(* CoDeSys 2.3.9.41 project: pogonazh_134_03_R.pro *)
(* Libraries: Util.lib 15.6.21 11:37:35, ПЛК_ПЧВ_v2.lib 17.6.21 09:07:23, STANDARD.LIB 15.6.21 11:37:35, IECSFC.LIB 15.6.21 11:37:35, ANALYZATION.LIB 15.6.21 11:37:35 *)

(* PLC configuration (modules and I/O channels)
InputByte AT %IB0.0 [ByteInput] 8 discrete inputs
DO_1_0 AT %QX1.0 [BitOutput] First
DO_1_1 AT %QX1.1 [BitOutput] Second
DO_2_0 AT %QX2.0 [BitOutput] First
AT %QX2.1 [BitOutput] Second
DO_3_0 AT %QX3.0 [BitOutput] First
DO_3_1 AT %QX3.1 [BitOutput] Second
DO_4_0 AT %QX4.0 [BitOutput] First
DO_4_1 AT %QX4.1 [BitOutput] Second
DO_5_0 AT %QX5.0 [BitOutput] First
DO_5_1 AT %QX5.1 [BitOutput] Second
DO_6_0 AT %QX6.0 [BitOutput] First
DO_6_1 AT %QX6.1 [BitOutput] Second
AT %QX7.0 [BitOutput] Special output
modbusLastAddr AT %QD8.0 [DWordOutput] Last address
modbusLastErr AT %QW8.1 [WordOutput] Last error
RS-485-1 [COM1_USART] node 0, in %IB8.0 out %QB8.0 {CommunicationSpeed = 19200; Parity = NO PARITY CHECK; BitLength = 8 bits; StopLength = One stop bit; InterfaceType = RS485; FrameOriented = RTU; Timeout = 0; Visibility = No}
Universal Modbus device [ID2000] node 1, in %IB8.1 out %QB8.1 {ModuleIP = 10:0:0:223; ServiceTimeout = 150; TCPport = 502; NetMode = Serial; ModuleSlaveAddress = 2; RequestType = By poll time; PeriodOfService = 1000; Visibility = No; RepeatCounter = 2; ByteSequence = Native}
  AT %QB8.1.0 [ComChannel] Command (0xff - Start)
Dist_on_pistol_1 AT %IW8.1.0.0 [WordInput]
Dist_on_pistol_2 AT %IW8.1.1.0 [WordInput]
Dist_on_pistol_3 AT %IW8.1.2.0 [WordInput]
Dist_on_pistol_4 AT %IW8.1.3.0 [WordInput]
Dist_on_pistol_5 AT %IW8.1.4.0 [WordInput]
Dist_on_pistol_6 AT %IW8.1.5.0 [WordInput]
Dist_off_pistol_1 AT %IW8.1.6.0 [WordInput]
Dist_off_pistol_2 AT %IW8.1.7.0 [WordInput]
Dist_off_pistol_3 AT %IW8.1.8.0 [WordInput]
Dist_off_pistol_4 AT %IW8.1.9.0 [WordInput]
Dist_off_pistol_5 AT %IW8.1.10.0 [WordInput]
Dist_off_pistol_6 AT %IW8.1.11.0 [WordInput]
DistOnPistMinimum AT %IW8.1.12.0 [WordInput]
qInvStatusW AT %QW8.1.13.0 [WordOutput]
AT %QB8.2.0 [ComChannel] Command (0xff - Start)
iTP1 AT %IW8.2.0.0 [WordInput]
iTP2 AT %IW8.2.1.0 [WordInput]
iTP3 AT %IW8.2.2.0 [WordInput]
iTP4 AT %IW8.2.3.0 [WordInput]
iTP5 AT %IW8.2.4.0 [WordInput]
iTP6 AT %IW8.2.5.0 [WordInput]
iTPGlob AT %ID8.2.6.0 [FloatInput]
iDate AT %ID8.2.7.0 [FloatInput]
qDate AT %QD8.2.8.0 [FloatOutput]
AT %QB8.3.0 [ComChannel] Command (0xff - Start)
task_speed_panel_real AT %ID8.3.0.0 [FloatInput]
speed_at_50Hz AT %ID8.3.1.0 [FloatInput]
speed_at_25Hz AT %ID8.3.2.0 [FloatInput]
speed_Max_panel AT %ID8.3.3.0 [FloatInput]
speed_Min_panel AT %ID8.3.4.0 [FloatInput]
qDetR AT %ID8.3.5.0 [FloatInput]
qMetR AT %ID8.3.6.0 [FloatInput]
follow_Sign_Loss AT %IW8.3.7.0 [WordInput]
qMaxDetLen AT %IW8.3.8.0 [WordInput]
qVersion AT %QD8.3.9.0 [FloatOutput]
iPwd AT %IW8.3.10.0 [WordInput]
AT %QB8.4.0 [ComChannel] Command (0xff - Start)
qInputB_DO1_6 AT %QW8.4.0.0 [WordOutput]
AT %QB8.5.0 [ComChannel] Command (0xff - Start)
qStatusW AT %QW8.5.0.0 [WordOutput]
controlPing AT %ID8.5.1.0 [FloatInput]
qDet_met AT %QD8.5.2.0 [FloatOutput]
qDet_Cnt AT %QD8.5.3.0 [FloatOutput]
controlPong AT %QD8.5.4.0 [FloatOutput]
qAbuseW AT %IW8.5.5.0 [WordInput]
qlast_Det_Len AT %QD8.5.6.0 [FloatOutput]
qlast_Det_Time AT %QD8.5.7.0 [FloatOutput]
AT %QB8.6.0 [ComChannel] Command (0xff - Start)
Status_word AT %IW8.6.0.0 [WordInput]
Frequency AT %IW8.6.1.0 [WordInput]
Power AT %IW8.6.2.0 [WordInput]
Voltage AT %IW8.6.3.0 [WordInput]
Current AT %IW8.6.4.0 [WordInput]
Inv_Error AT %ID8.6.5.0 [DWordInput]
Minimum_frequency AT %IW8.6.6.0 [WordInput]
Maximum_frequency AT %IW8.6.7.0 [WordInput]
Command_word AT %QW8.6.8.0 [WordOutput]
Task_RS485 AT %IW8.6.9.0 [WordInput]
Set_Speed AT %QW8.6.10.0 [WordOutput] 0-16384
Set_MinTask AT %QD8.6.11.0 [DWordOutput]
Set_MaxTask AT %QD8.6.12.0 [DWordOutput]
*)

(* Task configuration *)
TASK cycle_counters (PRIORITY := 0); (* freewheeling *)
	counters();
END_TASK
TASK main_task (PRIORITY := 1); (* freewheeling *)
	PLC_PRG();
END_TASK

(* Global variable list: Global_Variables *)
VAR_GLOBAL
	details_meters: REAL;			(*прошло деталей в метрах - берётся от длины в мм*)
	contr_StatusW:  WORD;   			(*статусное слово контроллера - заполняем в главном цикле*)
	contr_AbuseW: WORD;			(*командное слово контроллера - отрабатывает в главном цикле*)
       needSynhro : BOOL := TRUE;	(*Если требуется синхронизация - конвейер не обрабатывает команды управления*)
	freeCounters: BOOL := TRUE;	(*приказ очистить массив счетчика и ВЫКЛючить Пистолеты*)
	doBlur: BOOL := FALSE;			(*приказ делать сглаживание на сенсоре*)
	last_Det_length: REAL := 0.0;
	version: REAL := 0.3;
END_VAR

VAR_GLOBAL   (*переменные ошибок*)
	errSensor_stick: BOOL := FALSE; (*залипание*)
	errSensor_bounce: BOOL := FALSE; (*дребезг*)
	CALC_DET_LEN: REAL; 			(* накопитель для выработки ошибки *)
	errSensor_Glob: BOOL := FALSE; (* вырабатывается если количество деталей превысило максимум
											или слишком длинная деталь - ошибки находятся в разных переменных это их сумма
											пока активна ошибка - не будут накапливаться данные о деталях, пистолеты выключатся*)
	errTaskSpeed: BOOL := FALSE; 	(* вырабатывается если значение скорости не в диапазоне макс/мин или равно 0 *)

END_VAR

VAR_GLOBAL
	(*Входы контроллера*)
	Start_conveyor: BOOL;    			(*DI_1 Включить конвейер *)
	Stop_conveyor: BOOL;   			(*DI_2 Выключить конвейер *)
	Following_machine: BOOL;   		(*DI_3 Сигнал от следующей машины*)
	Fan_on: BOOL;					(*DI_4 Вытяжка включена*)
	Door_Closed: BOOL;				(*DI_5 Концевой выключатель двери*)
	Limit_switch_part: BOOL;			(*DI_6 Концевой выключатель наличия детали*)
(*	Pistols_5_8_run: BOOL;			(*DI_7 Включены пистолеты 5-8*) нет в проекте. всего 6*)

	(*Выходы контроллера*)
	Conveyor_green: BOOL;                     (*Конвейер готов к включению (сигнальная лампа) *)
	Conveyor_runNow: BOOL;			(*Конвейер поехал,сигнал на предыдущую машину *)

END_VAR

VAR_GLOBAL RETAIN PERSISTENT (*эти данные хранятся в энергонезависимой памяти*)
	details_count: REAL;				(*Счётчик кол-ва деталей. Сбрасывается по команде с панели *)
	details_mMeters: REAL;			(*Счётчик общей длины детали в мм, сбрасывается с панели *)
	details_Real_mMeters: REAL;	(*Необнуляемый счётчик  общей длины детали в мм*)
END_VAR

(* POU counters, ST *)
PROGRAM counters
VAR CONSTANT
	DETCNT: INT := 12;
	PISTCNT: INT := 6;
	PISTADD : INT := 2; (* mm !!!*)
	t0 : TIME := t#0ms;
END_VAR

VAR
	PistLen: ARRAY[1..PISTCNT,0..1] OF REAL;        (* 0 - Up Len, 1 - Off Len *)
	PistTime: ARRAY[1..PISTCNT] OF REAL;        (*iTP1,.. iTP5,.. *)
	PIST: ARRAY[1..PISTCNT] OF BOOL;
	DET: ARRAY[0..DetCNT,0..1] OF TIME; (* ЗАПОЛНЯЕТСЯ СПРАВА,  движется влево.  0 - начало жизни; 1 - конец детали, если конец = 0 - ещё не кончилась*)
	i,j: INT;
	detOn: BOOL;
	detOff: BOOL;
	need_Pistols_On : BOOL;
	SPEED : REAL; (* mm / ms *)
	CyclLEN: REAL; (* mm *)
	last_Det_time: TIME;
	cycleinterval_ms_calc: REAL;
	T, lastTime: TIME;
	rl, rlH, rlT: REAL;
	rl_TPGlob: REAL;
	MaxPIST: REAL;
	tt: TIME;
	last_Limit_switch_part: BOOL;
	partBlur: BLUR_6;
	err: BOOL;
END_VAR
need_Pistols_On := FALSE;

T := TIME();
cycleinterval_ms_calc := TIME_TO_REAL(T-lastTime)+0.0;
lastTime := T;

SPEED := task_speed_panel_real / 60.0;
CYCLLEN := SPEED * cycleinterval_ms_calc;

	(*Концевой выключатель наличия детали причём если нет его ошибки*)
partBlur(IN := DI_6 AND NOT errSensor_glob, EN := doBlur, Q => Limit_switch_part);
(*Pistols_5_8_run:=DI_7; 	(*Включены пистолеты 5-8*) нет в проекте. всего 6 пистолетов одновременно*)

detOn := FALSE;
detOff := FALSE;

IF NOT last_Limit_switch_part AND Limit_switch_part THEN (*деталь началась*)
	detOn := TRUE;
	last_Det_length := 0.0;
	last_Det_time := T;
	CALC_DET_LEN := 0.0;
END_IF;

IF last_Limit_switch_part AND NOT Limit_switch_part THEN (*деталь прошла*)
	details_count := details_count +1;
	qLast_Det_time := TIME_TO_REAL(T-last_Det_time);
	detOff := TRUE;
END_IF;

(*запомнить состояние датчика*)
last_Limit_switch_part := Limit_switch_part;

(* если сенсор включен - накопить ошибку *)
IF Limit_switch_part THEN
   CALC_DET_LEN := CALC_DET_LEN + CyclLEN;
END_IF;

IF (qmaxDetLen > 0) AND (CALC_Det_LEN > qmaxDetLen) THEN
	errSensor_stick := TRUE;
END_IF;

(* заполнить массив включения выключения если не синхронизация *)
IF NOT needSynhro THEN
   PistLen[1,0] := Dist_on_pistol_1; PistLen[1,1] := Dist_off_pistol_1+PISTADD;
   PistLen[2,0] := Dist_on_pistol_2; PistLen[2,1] := Dist_off_pistol_2+PISTADD;
   PistLen[3,0] := Dist_on_pistol_3; PistLen[3,1] := Dist_off_pistol_3+PISTADD;

	PISTTime[1] := iTP1;
	PISTTime[2] := iTP2;
	PISTTime[3] := iTP3;

   PistLen[4,0] := Dist_on_pistol_4; PistLen[4,1] := Dist_off_pistol_4+PISTADD;
   PistLen[5,0] := Dist_on_pistol_5; PistLen[5,1] := Dist_off_pistol_5+PISTADD;
   PistLen[6,0] := Dist_on_pistol_6; PistLen[6,1] := Dist_off_pistol_6+PISTADD;
	PISTTime[4] := iTP4;
	PISTTime[5] := iTP5;
	PISTTime[6] := iTP6;

END_IF;

MaxPIST := 0;						(*расстояние смерти детали - последняя точка где могут покрасить*)
FOR i := 1 TO PISTCNT DO
   MaxPIST := MAX(PistLen[i,0] + PistLen[i,1], MaxPist);
END_FOR;
MaxPIST := MaxPIST + 100; (*!!! добавим 10 см *)

(* ================================ ПОНЕСЛОСЬ ДЕТАЛИ ============================= *)

(* нахуй пистолеты *)
FOR j := 1 TO PISTCNT DO
   pist[j] := FALSE;
END_FOR;

IF NOT ErrSensor_glob AND NOT FreeCounters THEN   (* ---------------------------------------  далее делаем все действия если нет ошибки сенсора *)

(* деталь приехала, сместить все детали налево если первая не нолик *)
IF DetOn THEN
	IF DET[DETCNT,0] > t0 THEN
		FOR i:= 0 TO DETCNT-1  DO
			DET[i,0] := DET[i+1,0];
			DET[i,1] := DET[i+1,1];
		END_FOR;
	END_IF;
	DET[DETCNT,0] := T;
	DET[DETCNT,1] := t0; (* начала набирать время *)
	(*проверить, если в индекс 0 попала деталь, живая ещё, значит ошибка сенсора или другие проблемы *)
	IF DET[0,0] > t0 THEN
		ErrSensor_bounce := TRUE;
	END_IF;
END_IF;

(* деталь ПРОехала*)
IF DetOff AND (DET[DETCNT,0] > t0) THEN
	DET[DETCNT,1] := T;
       (* увеличим погонаж*)
	rl := TIME_TO_REAL(DET[DETCNT,1]-DET[DETCNT,0])*SPEED;		(*длина детали в мм*)
	(* проверка на длину детали, принятие решения*)
	IF rl < 20.0 THEN (*детали меньше 20 мм - не считово*)
		DET[DETCNT,0] := t0;
		DET[DETCNT,1] := t0;
	ELSE
		details_mMeters := details_mMeters + rl ;
		details_Real_mMeters := details_Real_mMeters + rl;
		last_Det_Length := rl;
	END_IF;
END_IF;

(* зажжём пистолеты *)

(* сперва убьём плохие детали*)
FOR i := 1 TO DETCNT DO
   IF DET[i,0] > t0 AND DET[i,1] > t0 THEN
	rlT := TIME_TO_REAL(T-DET[i,1])*SPEED; (*положение хвоста сейчас*);
	IF rlT > MaxPIST THEN (*условие убийства хвост укатил за максимальный пистолет + *)
		DET[i,0] := t0;
		DET[i,1] := t0;
	END_IF;
   END_IF;
END_FOR;

rl_TPGlob := iTPGlob;

FOR i := 1 TO DETCNT DO   (*пройдем по всем начиная с первой (1) деталям с начала до конца*)
IF DET[i,0] > t0 THEN (*деталь есть ?*)
	(*посмотрим на пистолеты*)
	FOR j := 1 TO PISTCNT DO
	IF NOT PIST[j] THEN (*если пистолет ещё не включен*)
		tt := DET[i,1];
		IF tt = t0 THEN tt := T; END_IF;
		rlH := (TIME_TO_REAL(T-DET[i,0])+PistTime[j]-rl_TPGlob )*SPEED; (*положение головы сейчас*);
		rlT := (TIME_TO_REAL(T-tt)+PistTime[j]/10-rl_TPGlob)*SPEED; (*положение хвоста сейчас  ! хвост ближе головы   ??? !!! div 10 - время выключения*);
		(*наконец зажжём факелы*)
		IF (MAX(PistLen[j,0], rlT) <= MIN(PistLen[j,0]+PistLen[j,1], rlH)) THEN
			PIST[j] := TRUE;
		END_IF;
	END_IF;
	END_FOR;
END_IF;
END_FOR;


need_Pistols_On := contr_abuseW.1  AND Door_Closed AND Fan_on; (*просит включить распыление и ВЫтяжка *)

ELSE (* т.е. если сенсор или надо очистить - очистить*)
	FOR i:= 0 TO DETCNT  DO
		DET[i,0] := t0;
		DET[i,1] := t0;
	END_FOR;
	FreeCounters := FALSE;
END_IF; (* ------------------------------------------ после проверки ошибки сенсора*)

(*включить/выключить пистолеты *)
DO_3_0 := pist[1] OR need_Pistols_On;
DO_3_1 := pist[2] OR need_Pistols_On;
DO_4_0 := pist[3] OR need_Pistols_On;
DO_4_1 := pist[4] OR need_Pistols_On;
(*DO_5_0 := pist[5] OR need_Pistols_On;
DO_5_1 := pist[6] OR need_Pistols_On; *)
END_PROGRAM

(* POU BLUR_6, ST *)
FUNCTION_BLOCK BLUR_6
VAR_INPUT
	IN,			(*вход для смягчения*)
	EN:BOOL;	(*если не разрешено, то Q равен IN, при этом ctr = 0*)
END_VAR
VAR_OUTPUT
	Q:BOOL;	(*Q := CTR > 2 (i.e. 3,4,5)*)
END_VAR
VAR
	CTR: INT;	(*0,1,2,3,4,5*)
END_VAR
IF NOT EN THEN
	Q := IN;
	CTR := 0;
ELSE
	IF in AND ctr<5 THEN ctr := ctr+1;END_IF;
	IF NOT in  AND ctr>0 THEN ctr := ctr-1;END_IF;
	Q := CTR > 2;
END_IF;
END_FUNCTION_BLOCK

(* POU PLC_PRG, ST *)
PROGRAM PLC_PRG
VAR
	synhroW: DWORD := 0;

	com_word: com_word_fb;
	Invertor_stop: BOOL := FALSE;
	Invertor_start: BOOL := FALSE;
	Invertor_reverse:BOOL := FALSE;
	Invertor_speed_ok: BOOL := FALSE;

(*переменные объединяющиес текущий статус контроллера*)
	Invertor_Pwr_On: BOOL := FALSE; (*инвертор найден по шине, получен статус отличный от 0 и он в автомате и готов*)
	Conveyor_On: BOOL; (*включен двигатель конвейера*)

(*просто какие-то временные переменные*)
	w1: WORD;
	dw, mit, mat: DWORD;
	bol: BOOL;
	b: REAL;
	k: REAL;
	modbusInvLastErr: WORD := 0;
	ispwdok: pwdOk
;
(* Статус частотника *)
	stat_word: stat_word_fb;

	Invertor_alarm: BOOL;		(* Авария частотника *)
	Invertor_warning: BOOL; 		(* Предупреждение частотника *)
	Invertor_auto: BOOL;			(* Частотник в автоматическом режиме *)
	Invertor_work: BOOL; 			(* Частотник в работе *)

(*переменные для управления ПЧВ*)
	rsp : REAL;
	abuse_50Hz: BOOL; (*принуждает ПЧВ запустить двигатель на 50 Hz*)
	abuse_25Hz: BOOL; (*принуждает ПЧВ запустить двигатель на 25 Hz*)
	abuse_20Hz: BOOL;
	frequency_Equal: BOOL := FALSE;
	lastFreqReqw: WORD := 0;
	task_invertor: task_fb;
	TONRun: TON;
	TPRun: TOF;
	Ctr20: INT;

(*FB logic*)

	Run:BOOL;
	Stop:BOOL;
	Common_Alarm: BOOL;
	R_TRIG: R_TRIG;
	F_TRIG: F_TRIG;
	F_TRIG1: F_TRIG;
	RS1: RS;

	Maintenance: BOOL;
	al_password: BOOL;
END_VAR
(*проверка связи по модбасу с ПЧВ Addr=1 *)
IF  modbusLastAddr = 1 THEN
	modbusInvLastErr := modbusLastErr;
END_IF;

(*Статус частотника*)
stat_word(
	stat_word:= Status_word,
	ready_engine=> ,
	ready_drvive=> ,
	slow_stop_stat=> ,
	alarm=>Invertor_alarm ,
	warning=> Invertor_warning,
	task_stat=>Invertor_speed_ok ,
	avt=>Invertor_auto ,
	over_range=> ,
	work_stat=>Invertor_work ,
	voltage=> ,
	current=> ,
	heat=> );

Invertor_Pwr_On := (Status_Word > 0) AND (modbusInvLastErr = 0) AND Invertor_auto AND NOT Invertor_alarm;

(*проверка пароля*)
ispwdOk(pwd := iPwd, cDate := iDate, Ok =>  al_password, fixdate => qDate);
al_password := NOT al_password;

Start_conveyor:=DI_1 ;	(*Включение конвейера*)
Stop_conveyor:=NOT DI_2 ; 	(*Отключение конвейера*)
Following_machine:=DI_3; (*Сигнал от предыдущей машины*)
Fan_on:=DI_4; 			(*Вытяжка включена*)
Door_closed := NOT DI_5; 		(*Дверь закрыта наоборот )) *)
(*Pistols_5_8_run := DI_7; (*выбраны 5-8 пистолеты*)*)
Maintenance := NOT Door_closed;

IF follow_Sign_Loss =2 THEN Following_machine := TRUE; END_IF;

errTaskSpeed :=  	(task_speed_panel_real <= 0) OR
					(speed_at_50Hz <= 0) OR
					(speed_at_50Hz <= speed_at_25Hz) OR
					(speed_Max_panel <= speed_Min_panel) OR
					(speed_Max_panel <= 0) OR
					(task_speed_panel_real > speed_Max_panel) OR
					(task_speed_panel_real < speed_Min_panel);

errSensor_bounce := errSensor_bounce OR  al_Password;
errSensor_Glob := errSensor_stick OR errSensor_bounce ;

Conveyor_On := Invertor_Work;

(*посчитаем - выставил ли частотник реальную частоту*)
w1 := (100*(100*Frequency+1)) / (100*lastFreqReqw+1);
frequency_Equal := Invertor_Work AND ((w1 > 97) OR Invertor_speed_ok);    (*скорость соответствует на 98% и более*)

(*программируем общую логику*)
(*надо получить состояние, зажечь лампу, дать сигнал на машину*)

(*работа зависит от    			 follow_Sign_Loss *)

IF NOT Maintenance THEN R_TRIG
(CLK:=Start_conveyor, 		(*Выделение переднего фронта на запуск конвейера*)
 Q=>Run );
END_IF;

TONRun(IN := Start_conveyor, PT:= T#4s);

R_TRIG
(CLK:=Stop_conveyor,			(*Выделение переднего фронта на останов конвейера*)
 Q=>Stop );

Common_Alarm := errSensor_glob OR errTaskSpeed OR Invertor_Alarm OR NOT Invertor_Pwr_On ;

RS1(
SET:= ( Fan_On AND Run  AND Invertor_Pwr_On AND Door_Closed),
RESET1:= (Stop OR NOT Fan_On OR NOT Door_Closed OR Common_alarm),
Q1=> Conveyor_green);

IF Conveyor_green THEN (*есть базовое разрешение на включение, проверим логику с ведомой машиной*)
   Conveyor_runNow := Following_machine; (*запустить конвейер по сигналу от след машины*)
IF follow_Sign_Loss > 0 THEN (*определено ждать*)
  ;
   (*помигаем лампочкой если нет машины*)
   (*мигать будем потом там внизу*)
ELSE (*определено закончить работу*)
   Conveyor_green := Following_machine;
END_IF;
ELSE (*конвейер не зелёный*)
   Conveyor_runNow := FALSE;
END_IF;

Invertor_start:=Conveyor_runNow;

(*задний фронт на останов частотника используем для обнуления массива*)
F_TRIG1(
	CLK:=Conveyor_runNow ,
	Q=> Invertor_stop);

IF abuse_20Hz OR (Conveyor_green AND NOT Following_machine) THEN (*замигаем лампу*)
   DO_1_0 := TIME_TO_DWORD(TIME()) MOD 1000 > 500;
ELSE
    DO_1_0:=Conveyor_green;  (*сигнальная лампа*)
END_IF;
DO_2_0:=Conveyor_runNow;  (*Конвейер включен(,сигнал на предыдущую машину)*)

(* создание слова статуса контроллера*)

contr_statusW.0  := 1; (*контроллер под питанием*)
contr_statusW.1 := Invertor_Pwr_On;
contr_statusW.2 := Fan_On;
contr_statusW.3 := Conveyor_On;
contr_statusW.4 := Door_Closed;
contr_statusW.5 := Following_machine;
(*contr_statusW.6 := Pistols_5_8_run;*)
contr_statusW.7 := Conveyor_runNow;
contr_statusW.8 := errSensor_stick;
contr_statusW.9 := errTaskSpeed;
contr_statusW.10 := Invertor_Alarm;
contr_statusW.11 := errSensor_bounce;

(*Загрузить возможные переменные с подчиненных устройств
 и проверить контрольную сумму. предварительно её рассчитав.

выставит needSynhro - что означает не все данные загружены
требуется синхронизация!
*)

freeCounters := errSensor_glob OR NOT Door_Closed OR NOT fan_on OR Invertor_stop; (* если ошибка сенсора или дверь не закрыта -  очистить список деталей *)

synhroW :=
	Dist_on_pistol_1+Dist_off_pistol_1+
	Dist_on_pistol_2+Dist_off_pistol_2+
	Dist_on_pistol_3+Dist_off_pistol_3+
	Dist_on_pistol_4+Dist_off_pistol_4+
	Dist_on_pistol_5+Dist_off_pistol_5+
	Dist_on_pistol_6+Dist_off_pistol_6+
(*	Dist_on_pistol_7+Dist_off_pistol_7+
	Dist_on_pistol_8+Dist_off_pistol_8+
	Dist_on_pistol_9+Dist_off_pistol_9+*)
	follow_Sign_Loss+
	TRUNC(10*task_speed_panel_real)+
	TRUNC(10*speed_at_50Hz)+
	TRUNC(10*speed_Max_panel)+
	TRUNC(10*speed_Min_panel)+
	qMaxDetLen+
	DistOnPistMinimum+
	TRUNC(10*speed_at_25Hz)+
	BOOL_TO_WORD(doBlur)+
	iTP1+iTP2+iTP3+iTP4+iTP5+iTP6+(*iTP7+iTP8+iTP9+*)
	TRUNC(10*ABS(iTPGlob));


controlPong := DWORD_TO_REAL(synhroW);
needSynhro :=  controlPing <> controlPong; (* установить необходимость синхронизации*)

contr_abuseW := qAbuseW;
needSynhro := needSynhro OR contr_abuseW.0; (*проверить не прислала ли панелька своё требование синхронизации*)

IF contr_abuseW.2 THEN (*bit 2 просит обнулить счётчики*)
	Details_Count := 0;
	Details_mMeters := 0;
END_IF;
IF contr_abuseW.3 THEN (*bit 3 просит установить счётчики*)
	Details_Count := qDetR;
	Details_mMeters := qMetR*1000;
END_IF;
IF contr_abuseW.4 THEN (*bit 4 просит сбросить ошибки*)
	errSensor_stick := FALSE;       (* сбросим ошибку сенсора, мало ли .... исправит ситуацию*)
	errSensor_bounce := FALSE;       (* сбросим ошибку сенсора, мало ли .... исправит ситуацию*)
	CALC_DET_LEN := 0.0;	(*сброс накопителя ошибки залипание*)
END_IF;
abuse_50Hz := contr_abuseW.5; (*bit 5 установить скорость 50 Hz*)
abuse_25Hz := contr_abuseW.6; (*bit 6 установить скорость 25 Hz*)
doBlur := contr_abuseW.7; (*bit 7 приказ делать сглаживание*)

TPRun(IN := FALSE);
IF Maintenance AND TONRun.Q OR NOT tpRun.Q THEN
   IF Ctr20 > 0 THEN Ctr20 := ctr20-1; END_IF;
  TPRun(IN := TRUE, PT := T#1s);
   IF TONRun.Q THEN Ctr20 := 600; END_IF; (* 600 = 10 min *)
END_IF;

IF stop OR door_closed THEN ctr20 := 0; END_IF;

abuse_20Hz := Maintenance AND (ctr20 > 0);

(* заполнить основные переменные для передачи в панельки.
передача 3 раза в сек *)

details_meters := details_mMeters / 1000;

qStatusW := contr_StatusW;
qDet_Cnt := Details_Count;
qDet_Met := Details_Meters;
qLast_det_len := last_Det_Length;
qInvStatusW := status_word;

w1 := SHL(InputByte,8);
w1.0 := DO_1_0;
w1.1 := DO_2_0;
w1.2 := DO_3_0;
w1.3 := DO_3_1;
w1.4 := DO_4_0;
w1.5 := DO_4_1;
w1.6 := DO_5_0;
w1.7 := DO_5_1;

w1.8 := frequency_Equal; (*!!! ??? was W1.6*)
qInputB_DO1_6 := w1;
qVersion := Version;

(*программируем ПЧВ*)
(*проверяем на ошибки и если всё ок - начинаем им управлять*)
	w1 := Task_RS485; (*0-16384*)

	IF NOT errTaskSpeed AND NOT needSynhro THEN (*вычисляем какую скорость поставить*)
		(*запрограммируем линейность по 2 точкам   ??? *)
		k := (50-25) / (speed_at_50Hz - speed_at_25Hz);
		b := 50-k*speed_at_50Hz;
		rsp := task_speed_panel_real * k + b; (*???*) (*rsp = необходимая частота Hz*)
		(*предыдущая версия расчёта по 1 коэффициенту*)
(*		rsp := task_speed_panel_real / speed_at_50Hz * 50; (*rsp = необходимая частота Hz*) *)

		w1 := REAL_TO_WORD(rsp*10); (*w1 теперь соответсвует частоте * 10 как и в мин, макс*)
		IF w1 < Minimum_frequency THEN w1 := Minimum_frequency; END_IF;
		IF w1 > Maximum_frequency THEN w1 := Maximum_frequency; END_IF;
		(*Maximum_frequency (*650   = 65Гц*)*)
		lastFreqReqw := w1;
		(*на этом этапе w1 : [0..650] НАДО конвертнуть в 0 - 16384*)
		rsp := 16384 * w1 / Maximum_frequency;
		w1 := REAL_TO_WORD(rsp);
	END_IF;
	IF errTaskSpeed AND NOT needSynhro THEN
		invertor_Start := FALSE;
	END_IF;

	bol := FALSE;
	IF NOT needSynhro AND (abuse_50Hz OR abuse_25Hz OR abuse_20Hz) THEN (*принудим двигатель раскрутиться на 50 hz*)
		w1 := 500;
		IF abuse_25Hz THEN w1 := 250; END_IF;
		IF abuse_20Hz THEN w1 := 200; END_IF;
		lastFreqReqw := w1;
		(*на этом этапе w1 = 500|250  НАДО конвертнуть в 0 - 16384*)
		rsp := 16384 * w1 / Maximum_frequency;
		w1 := REAL_TO_WORD(rsp);
		bol := (w1 > 0);
	END_IF;
       Set_MinTask := Minimum_frequency * 100;
	Set_MaxTask := Maximum_frequency * 100;
	Set_Speed := w1; (*0-16384*)


(*task_invertor(
	t_min:=task_frequency_min ,
	t_max:=task_frequency_max ,
	task_value:=task_frequency_invertor ,
	pre_task_value1:= ,
	pre_task_value2:=,
	pre_task_value3:= ,
	pre_task_value4:= ,
	num_task:= ,
	lim_h:= ,
	Idc_stop_val:= ,
	rs_off:= ,
	task_min=>mit ,
	task_max=>mat,
	task=>w1 ,
	pre_task_value=> ,
	pre_task_num=> ,
	lim_high=> ,
	Idc_stop=> ,
	rs_out=> );
*)
(*запустить двигатель*)
com_word(
	pre_task_num:= ,
	dc_stop:= ,
	slow_stop:=Invertor_stop ,
	fast_stop:= ,
	start:= Invertor_start OR bol,
	REVERSE:=FALSE ,
	com_word=>Command_word );
END_PROGRAM

(* POU pwdOk, ST *)
FUNCTION_BLOCK pwdOk
VAR_INPUT
	pwd: WORD;
	cDate: REAL;
END_VAR
VAR_OUTPUT
	ok: BOOL;
	fixdate: REAL;
END_VAR
VAR
END_VAR
CASE pwd OF
	27572: fixdate := 70.12; (*мастер пароль*)
	49646: fixdate := 21.01;
	17449: fixdate := 21.02;
	48854: fixdate := 21.03;
	21865: fixdate := 21.04;
	44836: fixdate := 21.05;
	43462: fixdate := 21.06;
	53980: fixdate := 21.07;
	52141: fixdate := 21.08;
	17184: fixdate := 21.09;
	27117: fixdate := 21.10;
	35262: fixdate := 21.11;
	62814: fixdate := 21.12;
ELSE
			fixdate := 00.00;
END_CASE;
ok := cDate <= fixDate;
END_FUNCTION_BLOCK
